FUNCTION_BLOCK Q_Attribute_AUDI (* Command change attribute( Part 6 - F.38 ) *)
  (* Standard: ISO 11783-6; Description: Copyright (c) 2022 HR Agrartechnik GmbH This program and the accompanying materials are made available under the terms of the Eclipse Public License 2.0 which is available at https://www.eclipse.org/legal/epl-2.0/ SPDX-License-Identifier: EPL-2.0 see Description Tab *)
  (* Version 1.0, 2025-02-23, Franz Höpfinger, HR Agrartechnik GmbH *)
  PACKAGE isobus::UT::Q;
  IMPORT isobus::UT::Q::const::IDs::ID_NULL;
  (* Documentation:
  Command change attribute( Part 6 - F.38 )
   This command is used to change any attribute with an assigned AID. This message cannot be used to change strings. This FB wraps isobus::UT::Q::Q_Attribute and addresses two distinct parameters — u16ObjId (the object whose attribute is changed) and u8IdAttribute (the Attribute ID, AID).
   Valid values for u16ObjId (the object whose attribute is changed)
   A change-attribute Object ID is valid if it falls within one of the following ISO 11783-6 ID ranges (Annex F.38):
    - DataMask: 1000 – 1999
   - AlarmMask: 2000 – 2999
   - SoftKeyMask: 4000 – 4999
   - Key: 5000 – 5999
   - Button: 6000 – 6999
   - InputBooleanField: 7000 – 7999
   - InputStringField: 8000 – 8999
   - InputNumberField: 9000 – 9999
   - InputListField: 10000 – 10999
   - AuxiliaryFunctionType2: 31000 – 31999
    Valid values for u8IdAttribute (AID)
   The Attribute ID (AID) selects which attribute of the addressed object is changed. Valid AIDs are object-type specific and are defined in ISO 11783-6 Annex B, in the attribute table of each object type. An AID with no attribute assigned is rejected by the VT (F.39, bit 1 = Invalid Attribute ID).
   ID_NULL (65535) is not a command target but can be used in INIT to deactivate the FB. Any ID outside these ranges is invalid for commanding.
   param[in] {u16ObjId, uint16_t}
   Object ID
   param[in] {u8IdAttribute, uint8_t}
   Attribute ID (AID) - see description of wished object
   param[in] {u32ValueAttribute, uint32_t}
   New value for attribute
   Return Values: 
   int16_t
    - VT_E_NO_ERR (0) - OK
   - VT_E_OVERFLOW (-6) - buffer overflow
   - VT_E_NOACT (-8) - Command not possible in current state
   - VT_E_NO_INSTANCE (-21) - No VT client available
   - VT_E_ISO_INSTANCE_INVALID (-129) - Identifier for instance (connection) invalid
   - VT_E_NOT_ALIVE (-130) - Identifier for instance valid, but VT Dead.
  *)
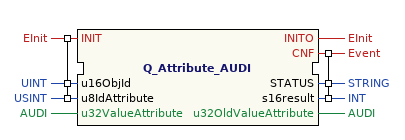
  EVENT_INPUT
    INIT : EInit WITH u16ObjId, u8IdAttribute; (* Service Initialization *)
  END_EVENT
  EVENT_OUTPUT
    INITO : EInit; (* Initialization Confirm *)
    CNF WITH STATUS, s16result; (* Confirmation of Requested Service *)
  END_EVENT
  VAR_INPUT
    u16ObjId : UINT := ID_NULL; (* Object ID *)
    u8IdAttribute : USINT; (* Attribute ID (AID) - see description of wished object *)
  END_VAR
  VAR_OUTPUT
    STATUS : STRING; (* Service Status *)
    s16result : INT; (* retval see description *)
  END_VAR
  SOCKETS
    u32ValueAttribute : adapter::types::unidirectional::AUDI; (* New value for attribute *)
  END_SOCKETS
  PLUGS
    u32OldValueAttribute : adapter::types::unidirectional::AUDI; (* Old value for attribute *)
  END_PLUGS
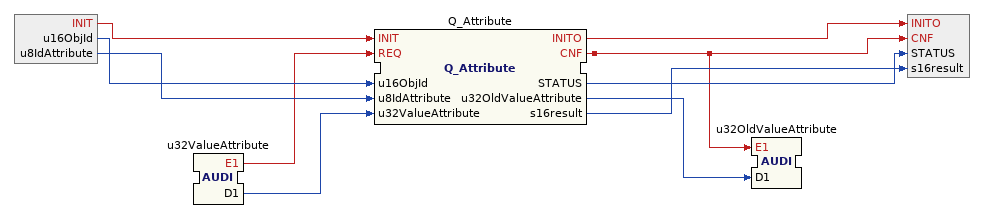
  FBS
    Q_Attribute : isobus::UT::Q::Q_Attribute;
  END_FBS
  EVENT_CONNECTIONS
    INIT TO Q_Attribute.INIT;
    Q_Attribute.INITO TO INITO;
    Q_Attribute.CNF TO CNF;
    u32ValueAttribute.E1 TO Q_Attribute.REQ;
    Q_Attribute.CNF TO u32OldValueAttribute.E1;
  END_CONNECTIONS
  DATA_CONNECTIONS
    Q_Attribute.STATUS TO STATUS;
    u16ObjId TO Q_Attribute.u16ObjId;
    u8IdAttribute TO Q_Attribute.u8IdAttribute;
    u32ValueAttribute.D1 TO Q_Attribute.u32ValueAttribute;
    Q_Attribute.u32OldValueAttribute TO u32OldValueAttribute.D1;
    Q_Attribute.s16result TO s16result;
  END_CONNECTIONS
END_FUNCTION_BLOCK
